// TIA Portal project "PLC_Batt" (V16)

(* hardware
DEVICE "S71500/ET200MP station_1"  S7-1500 station
   slot 0: "Rail_0"  Rack  6ES7 590-1***0-0AA0
   slot 1: "PLC_1"  CPU 1516-3 PN/DP  6ES7 516-3AN02-0AB0  V2.8
      slot 3: "CPU display_1"  6ES7591-1BA00-0AA0
      slot 32768: "PROFINET interface_1"  X1
      slot 33024: "PROFINET interface_2"  X2
      slot 33280: "DP interface_1"  X3
      slot 34817: "Virtual CP interface port_1"  Virtual CP interface port  Virtual CP interface port
DEVICE "HMI_1"  KTP700 Basic PN
   slot 0: "HMI_1"  KTP700 Basic PN  6AV2 123-2GB03-0AX0  16.0.0.0
   slot 1: "HMI_RT_1"  KTP700 Basic PN  6AV2 123-2GB03-0AX0  16.0.0.0
   slot 5: "HMI_1.IE_CP_1"  PROFINET Interface  16.0.0.0
      slot 1: "PROFINET Interface_1"  PROFINET Interface
         slot 1: "Port_1"  Port
*)

// ===== PLC "PLC_1"  CPU 1516-3 PN/DP =====

VAR_GLOBAL   // PLC tag table "inputTags"
   "batteryTesterDetector" AT %I0.0 : Bool;
   "batteryVisionDetector" AT %I0.1 : Bool;
   "Clock_Byte" AT %MB0 : Byte;
   "Clock_10Hz" AT %M0.0 : Bool;
   "Clock_5Hz" AT %M0.1 : Bool;
   "Clock_2.5Hz" AT %M0.2 : Bool;
   "Clock_2Hz" AT %M0.3 : Bool;
   "Clock_1.25Hz" AT %M0.4 : Bool;
   "Clock_1Hz" AT %M0.5 : Bool;
   "Clock_0.625Hz" AT %M0.6 : Bool;
   "Clock_0.5Hz" AT %M0.7 : Bool;
END_VAR

VAR_GLOBAL   // PLC tag table "safetyTags"
   "safetyCurtain1" AT %I1.0 : Bool;
   "safetyCurtain2" AT %I1.1 : Bool;
   "safetyCurtain3" AT %I1.2 : Bool;
   "safetyCurtain4" AT %I1.3 : Bool;
   "safetyCurtain5" AT %I1.4 : Bool;
   "safetySwitch1" AT %I2.5 : Bool;
   "safetySwitch2" AT %I2.6 : Bool;
   "safetySwitch3" AT %I2.7 : Bool;
   "warnignLamp" AT %Q1.0 : Bool;
END_VAR

DATA_BLOCK "BattTester_DB1"   // DB1
{ S7_Optimized_Access := 'TRUE' }
VERSION : 0.1
// stored: InstanceOfName BattTester
"BattTester"
BEGIN
END_DATA_BLOCK

DATA_BLOCK "VisionSystem_DB"   // DB6
{ S7_Optimized_Access := 'TRUE' }
VERSION : 0.1
// stored: InstanceOfName VisionSystem
"VisionSystem"
BEGIN
END_DATA_BLOCK

DATA_BLOCK "hmiController_DB"   // DB7
{ S7_Optimized_Access := 'TRUE' }
VERSION : 0.1
// stored: InstanceOfName hmiController
"hmiController"
BEGIN
END_DATA_BLOCK

DATA_BLOCK "daneProcesowe"   // DB8
{ S7_Optimized_Access := 'TRUE' }
VERSION : 0.1
   VAR
      visionSystem : Bool := 1;
      electricTesterSystem : Bool := 1;
      awaria : Bool;
      state : Int;
   END_VAR
BEGIN
END_DATA_BLOCK

// folder: System blocks/Program resources

DATA_BLOCK "IEC_Timer_0_DB"   // DB2
{ S7_Optimized_Access := 'TRUE' }
AUTHOR : Simatic
FAMILY : IEC
NAME : IEC_TMR
VERSION : 1.0
// stored: InstanceOfName IEC_TIMER
"IEC_TIMER"
BEGIN
END_DATA_BLOCK

DATA_BLOCK "PLC_1_Connection_DB"   // DB3
{ S7_Optimized_Access := 'TRUE' }
AUTHOR : SIMATIC
FAMILY : MC7Plus
NAME : TC_IP_v4
VERSION : 1.0
// stored: InstanceOfName TCON_IP_v4
"TCON_IP_v4"
BEGIN
   ID := 1;
   InterfaceId := 64;
   LocalPort := 2000;
END_DATA_BLOCK

DATA_BLOCK "IEC_Timer_0_DB_3"   // DB10
{ S7_Optimized_Access := 'TRUE' }
AUTHOR : Simatic
FAMILY : IEC
NAME : IEC_TMR
VERSION : 1.0
// stored: InstanceOfName IEC_TIMER
"IEC_TIMER"
BEGIN
END_DATA_BLOCK

DATA_BLOCK "IEC_Timer_0_DB_4"   // DB11
{ S7_Optimized_Access := 'TRUE' }
AUTHOR : Simatic
FAMILY : IEC
NAME : IEC_TMR
VERSION : 1.0
// stored: InstanceOfName IEC_TIMER
"IEC_TIMER"
BEGIN
END_DATA_BLOCK

DATA_BLOCK "IEC_Counter_0_DB"   // DB12
{ S7_Optimized_Access := 'TRUE' }
AUTHOR : Simatic
FAMILY : IEC
NAME : CNTR
VERSION : 1.0
// stored: InstanceOfName IEC_COUNTER
"IEC_COUNTER"
BEGIN
END_DATA_BLOCK

DATA_BLOCK "zliczaniePakietowCTU"   // DB13
{ S7_Optimized_Access := 'TRUE' }
AUTHOR : Simatic
FAMILY : IEC
NAME : CNTR
VERSION : 1.0
// stored: InstanceOfName IEC_COUNTER
"IEC_COUNTER"
BEGIN
END_DATA_BLOCK

// folder: (top level)

FUNCTION_BLOCK "BattTester"   // FB1, LAD
{ S7_Optimized_Access := 'TRUE' }
VERSION : 0.1
   VAR_INPUT
      batteryActivation : Bool;
   END_VAR
   VAR_OUTPUT
      dischargeMosfet : Bool;
      errorCode : Byte;
      finish : Bool;
      impedanceOut : Real;
      testResult : Bool;
   END_VAR
   VAR
      state : Byte := 0;
      sumOfVoltages : ULInt;
      numberOfReadingsVolts : Int;
      voltageBeforeTest : Real;
      impedance : Real;
   END_VAR
   VAR_TEMP
      batteryVoltage : Real;
      freq_to_peroid : Real;
      peroidInt : Int;
      impedanceTime : Time;
      meaonOfVoltages : ULInt;
      diffBetweenVoltages : ULInt;
      current : ULInt;
   END_VAR
   VAR CONSTANT
      timeToStart : Time := T#2s;   // czas potrzebny do uruchomienia testu po wykryciu akumulatora
      BATT_WAIT : Byte := 0;
      BATT_TEST : Byte := 1;
      BATT_AFTER_TEST : Byte := 2;
      BATT_WAIT_TO_LEAVE : Byte := 3;
      BATT_ERROR : Byte := 6;
      IMPEDANCE_TEST_FREQ : Int := 1000;
      BATT_CUT_OFF_VOLTAGE : Real := 60.0;
      BATT_MIN_VOLTAGE : Real := 40.0;
      RESISTOR_VAL : Real := 500.0;
   END_VAR
   VAR_TEMP   // added for the SCL form of the ladder/FBD networks
      _w1 : Bool;
   END_VAR
BEGIN

REGION Network 1
   // odczyt napiecia pinow baterii
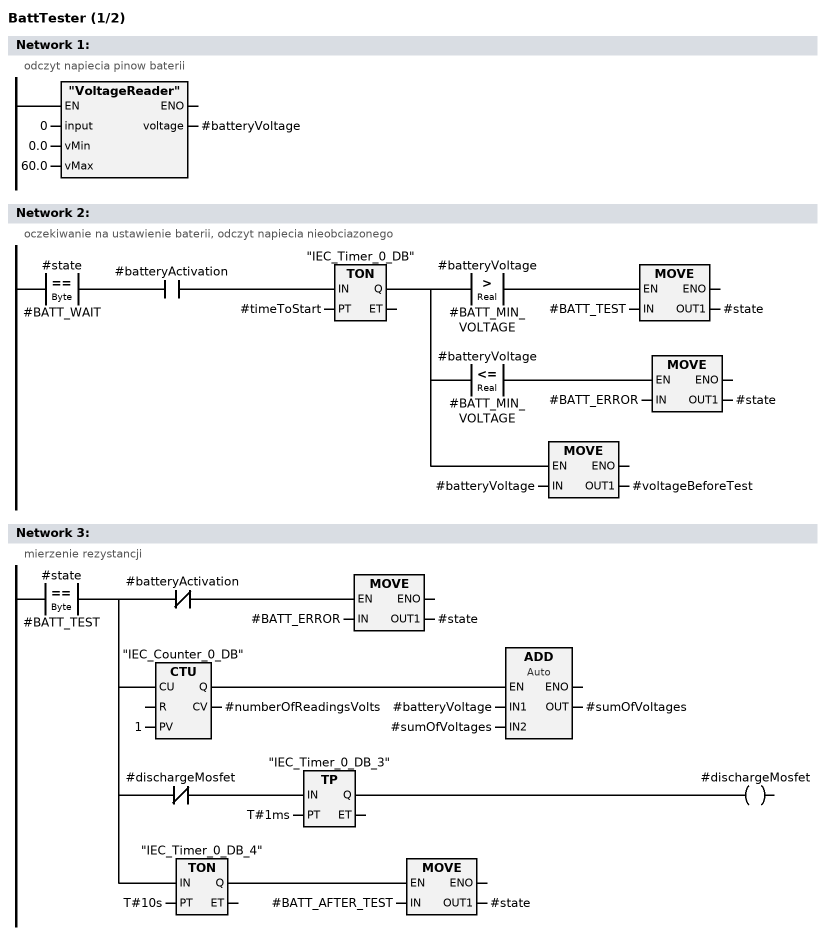
   RUNG wire#powerrail
      "VoltageReader"(input := 0, vMin := 0.0, vMax := 60.0, voltage => #batteryVoltage)
   END_RUNG
   // the same network as SCL:
   "VoltageReader"(input := 0, vMin := 0.0, vMax := 60.0, voltage => #batteryVoltage);
END_REGION

REGION Network 2
   // oczekiwanie na ustawienie baterii, odczyt napiecia nieobciazonego
   "IEC_Timer_0_DB".TON(IN := (#state = #BATT_WAIT) AND #batteryActivation, PT := #timeToStart);
   IF "IEC_Timer_0_DB".Q AND (#batteryVoltage > #BATT_MIN_VOLTAGE) THEN #state := #BATT_TEST; END_IF;
   IF "IEC_Timer_0_DB".Q AND (#batteryVoltage <= #BATT_MIN_VOLTAGE) THEN #state := #BATT_ERROR; END_IF;
   IF "IEC_Timer_0_DB".Q THEN #voltageBeforeTest := #batteryVoltage; END_IF;
END_REGION

REGION Network 3
   // mierzenie rezystancji
   #_w1 := #state = #BATT_TEST;
   IF #_w1 AND NOT #batteryActivation THEN #state := #BATT_ERROR; END_IF;
   "IEC_Counter_0_DB".CTU(CU := #_w1, PV := 1, CV => #numberOfReadingsVolts);
   IF "IEC_Counter_0_DB".Q THEN #sumOfVoltages := #batteryVoltage + #sumOfVoltages; END_IF;
   "IEC_Timer_0_DB_3".TP(IN := #_w1 AND NOT #dischargeMosfet, PT := T#1ms);
   #dischargeMosfet := "IEC_Timer_0_DB_3".Q;
   "IEC_Timer_0_DB_4".TON(IN := #_w1, PT := T#10s);
   IF "IEC_Timer_0_DB_4".Q THEN #state := #BATT_AFTER_TEST; END_IF;
END_REGION

REGION Network 4
   // wyznaczenie rezystancji wewnetrzenj ogniwa po tescie
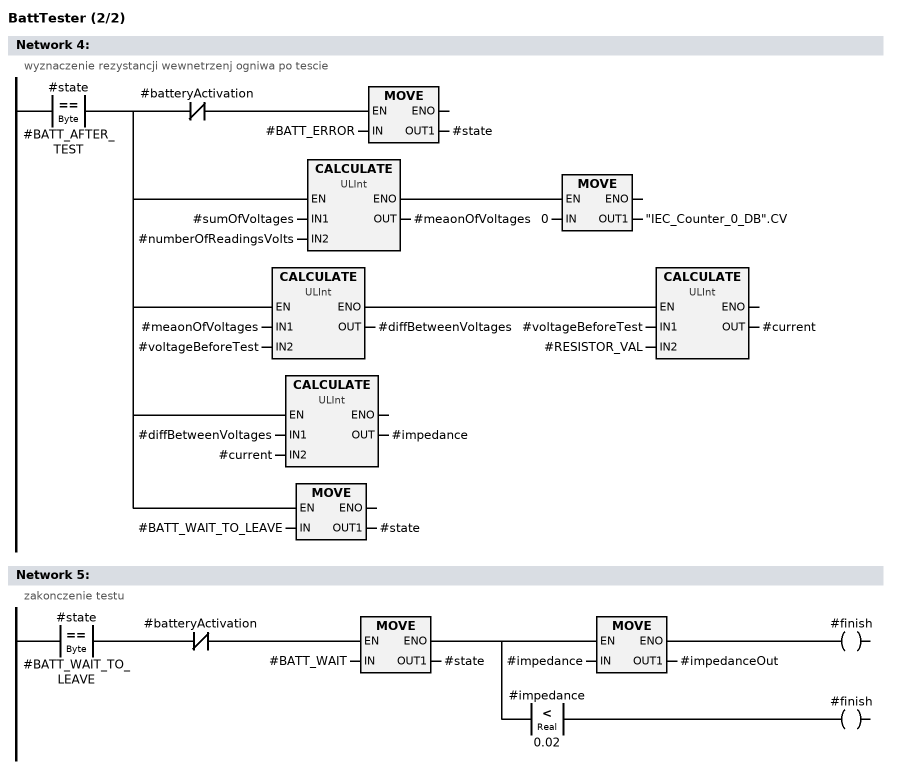
   RUNG wire#powerrail
      { S7_Templates := "SrcType := Byte" } EQ_Contact(in1 := #state, in2 := #BATT_AFTER_TEST)
      wire#w1
      I_Contact( #batteryActivation )
      Move(in := #BATT_ERROR, out1 => #state)
   END_RUNG
   RUNG wire#w1
      { S7_Templates := "SrcType := ULInt"; S7_Expression := "IN1/IN2" } Calculate(in1 := #sumOfVoltages, in2 := #numberOfReadingsVolts, out => #meaonOfVoltages)
      Move(in := 0, out1 => "IEC_Counter_0_DB".CV)
   END_RUNG
   RUNG wire#w1
      { S7_Templates := "SrcType := ULInt"; S7_Expression := "IN1 - IN2" } Calculate(in1 := #meaonOfVoltages, in2 := #voltageBeforeTest, out => #diffBetweenVoltages)
      { S7_Templates := "SrcType := ULInt"; S7_Expression := "IN1/IN2" } Calculate(in1 := #voltageBeforeTest, in2 := #RESISTOR_VAL, out => #current)
   END_RUNG
   RUNG wire#w1
      { S7_Templates := "SrcType := ULInt"; S7_Expression := "IN1 / IN2" } Calculate(in1 := #diffBetweenVoltages, in2 := #current, out => #impedance)
   END_RUNG
   RUNG wire#w1
      Move(in := #BATT_WAIT_TO_LEAVE, out1 => #state)
   END_RUNG
   // the same network as SCL:
   #_w1 := #state = #BATT_AFTER_TEST;
   IF #_w1 AND NOT #batteryActivation THEN #state := #BATT_ERROR; END_IF;
   IF #_w1 THEN
       #meaonOfVoltages := #sumOfVoltages/#numberOfReadingsVolts;
       "IEC_Counter_0_DB".CV := 0;
       #diffBetweenVoltages := #meaonOfVoltages - #voltageBeforeTest;
       #current := #voltageBeforeTest/#RESISTOR_VAL;
       #impedance := #diffBetweenVoltages / #current;
       #state := #BATT_WAIT_TO_LEAVE;
   END_IF;
END_REGION

REGION Network 5
   // zakonczenie testu
   RUNG wire#powerrail
      { S7_Templates := "SrcType := Byte" } EQ_Contact(in1 := #state, in2 := #BATT_WAIT_TO_LEAVE)
      I_Contact( #batteryActivation )
      Move(in := #BATT_WAIT, out1 => #state)
      wire#w1
      Move(in := #impedance, out1 => #impedanceOut)
      Coil( #finish )
   END_RUNG
   RUNG wire#w1
      { S7_Templates := "SrcType := Real" } LT_Contact(in1 := #impedance, in2 := 0.02)
      Coil( #finish )
   END_RUNG
   // the same network as SCL:
   #_w1 := (#state = #BATT_WAIT_TO_LEAVE) AND NOT #batteryActivation;
   IF #_w1 THEN
       #state := #BATT_WAIT;
       #impedanceOut := #impedance;
   END_IF;
   #finish := #_w1;
   #finish := #_w1 AND (#impedance < 0.02);
END_REGION
END_FUNCTION_BLOCK

FUNCTION_BLOCK "VisionSystem"   // FB2, LAD
{ S7_Optimized_Access := 'TRUE' }
VERSION : 0.1
   VAR_INPUT
      batteryDetection : Bool;
   END_VAR
   VAR_OUTPUT
      error : Bool;
      errorCode : Int;
      detectedFailedPacket : Bool;
      detectedGoodPacket : Bool;
      finished : Bool;
   END_VAR
   VAR
      TCON_Instance : TCON;
      state : Int := 1;
      batteryDetectionRisingEdge : Bool;
      recivedDataBatteryTest : Bool;
      test : Byte;
      disconnect : Bool;
      req : Bool := true;
      recv : Bool := false;
   END_VAR
   VAR_TEMP
      recivedData : Array[0..2] of Byte;
      recivedDataLen : Int;
      dataToSend : Array[0..2] of Byte;
   END_VAR
BEGIN

REGION Network 1
   // polaczenie z matlabem
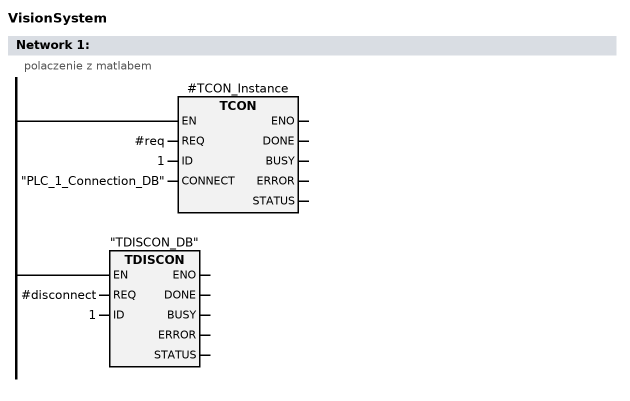
   #TCON_Instance(REQ := #req, ID := 1, CONNECT := "PLC_1_Connection_DB");   // TCON
   "TDISCON_DB"(REQ := #disconnect, ID := 1);   // TDISCON
END_REGION

REGION Network 2 (SCL)
   // maszyna stanu do testowania zgrzewów
   // maszyna stanu 
   CASE #state OF
       1: // oczekiwanie na baterie 
           IF #batteryDetection THEN
               #batteryDetectionRisingEdge := true;
               #state := 2; // zmiana stanu na 2
           END_IF;
       2: // wykryto baterie, wyslanie informacji do systemu wizyjnego 
           // wyslanie
           #dataToSend[0] := 5;
           #dataToSend[1] := 0;
           "TSEND_DB".TSEND(REQ:=TRUE,
                            ID:=1,
                            LEN:=2,
                            DATA:=#dataToSend);
           #state := 3;

       3: // odebranie i analiza odpowiedzi
           "TRCV_DB_1".TRCV(EN_R:=true,
                            ID:=1,
                            LEN:=2,
                            RCVD_LEN=>#recivedDataLen,
                            DATA:=#recivedData);
           IF #recivedDataLen > 0 THEN
               IF #recivedData[0] = 6 AND #recivedData[1] = 1 AND #finished = 0 THEN
                   #state := 4;
                   #detectedFailedPacket := 1;
                   #finished := 1;
               ELSE
                   #state := 4;
                   #detectedGoodPacket := 1;
                   #finished := 1;
               END_IF;
           END_IF;
       4: // oczekiwanie na opuszczenie baterii 
           #detectedFailedPacket := 0;
           #detectedGoodPacket := 0;
           IF #batteryDetection = false THEN
               #state := 1;
           END_IF;
   END_CASE;
END_REGION
END_FUNCTION_BLOCK

FUNCTION_BLOCK "hmiController"   // FB3, LAD
{ S7_Optimized_Access := 'TRUE' }
VERSION : 0.1
   VAR_INPUT
      batteryDetection : Bool;
      state : Int;
   END_VAR
   VAR_IN_OUT
      awaria : Bool;
   END_VAR
   VAR
      zliczaniePakietow : UDInt;
      pakietySprawne : UDInt;
      pakietyUszkodzone : UDInt;
      sprawnoscProcesu : Int;
      strState : String;
      uszkodzoneZgrzewy : UDInt;
      uszkodzoneOgniwa : UDInt;
   END_VAR
   VAR_TEMP
      awariaReset : Bool;
   END_VAR
BEGIN

REGION Network 1
   // zliczanie pakietow
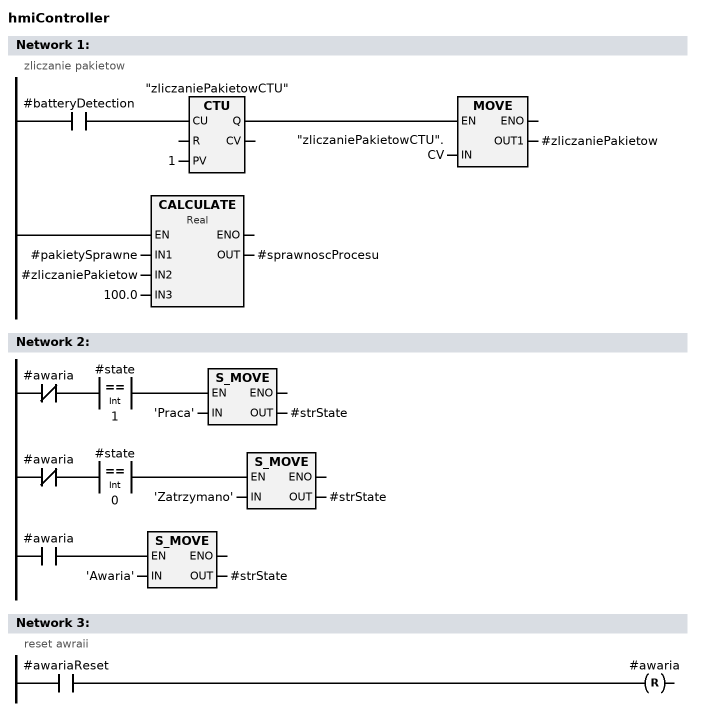
   "zliczaniePakietowCTU".CTU(CU := #batteryDetection, PV := 1);
   IF "zliczaniePakietowCTU".Q THEN #zliczaniePakietow := "zliczaniePakietowCTU".CV; END_IF;
   #sprawnoscProcesu := (#pakietySprawne / #zliczaniePakietow) * 100.0;
END_REGION

REGION Network 2
   RUNG wire#powerrail
      I_Contact( #awaria )
      { S7_Templates := "SrcType := Int" } EQ_Contact(in1 := #state, in2 := 1)
      S_Move(in := 'Praca', out => #strState)
   END_RUNG
   RUNG wire#powerrail
      I_Contact( #awaria )
      { S7_Templates := "SrcType := Int" } EQ_Contact(in1 := #state, in2 := 0)
      S_Move(in := 'Zatrzymano', out => #strState)
   END_RUNG
   RUNG wire#powerrail
      Contact( #awaria )
      S_Move(in := 'Awaria', out => #strState)
   END_RUNG
   // the same network as SCL:
   IF NOT #awaria AND (#state = 1) THEN #strState := 'Praca'; END_IF;
   IF NOT #awaria AND (#state = 0) THEN #strState := 'Zatrzymano'; END_IF;
   IF #awaria THEN #strState := 'Awaria'; END_IF;
END_REGION

REGION Network 3
   // reset awraii
   RUNG wire#powerrail
      Contact( #awariaReset )
      R_Coil( #awaria )
   END_RUNG
   // the same network as SCL:
   IF #awariaReset THEN #awaria := FALSE; END_IF;
END_REGION
END_FUNCTION_BLOCK

FUNCTION "VoltageReader" : Void   // FC1, LAD
{ S7_Optimized_Access := 'TRUE' }
VERSION : 0.1
   VAR_INPUT
      input : DInt;
      vMin : Real;
      vMax : Real;
   END_VAR
   VAR_OUTPUT
      voltage : Real;
   END_VAR
   VAR_TEMP
      tempVoltage : Real;
   END_VAR
BEGIN

REGION Network 1
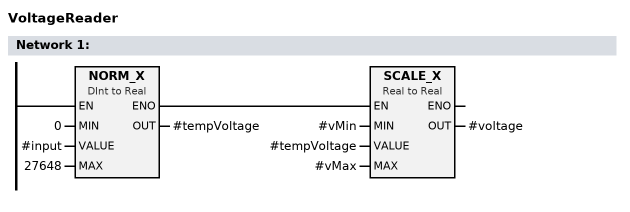
   RUNG wire#powerrail
      { S7_Templates := "[SrcType := DInt, DestType := Real]" } Normalize(min := 0, value := #input, max := 27648, out => #tempVoltage)
      { S7_Templates := "[SrcType := Real, DestType := Real]" } Scale(min := #vMin, value := #tempVoltage, max := #vMax, out => #voltage)
   END_RUNG
   // the same network as SCL:
   #tempVoltage := NORM_X(MIN := 0, VALUE := #input, MAX := 27648);
   #voltage := SCALE_X(MIN := #vMin, VALUE := #tempVoltage, MAX := #vMax);
END_REGION
END_FUNCTION

ORGANIZATION_BLOCK "Main"   // OB1, LAD, ProgramCycle
TITLE = "Main Program Sweep (Cycle)"
{ S7_Optimized_Access := 'TRUE' }
VERSION : 0.1
   VAR_INPUT
      Initial_Call : Bool;   // Initial call of this OB
      Remanence : Bool;   // =True, if remanent data are available
   END_VAR
   VAR_TEMP
      visionGoodBatt : Bool;
      visionFailBatt : Bool;
      finished : Bool;
   END_VAR
   VAR_TEMP   // added for the SCL form of the ladder/FBD networks
      _w1 : Bool;
      _w2 : Bool;
   END_VAR
BEGIN

REGION Network 1
   // system do testowania paramterów elektrycznych
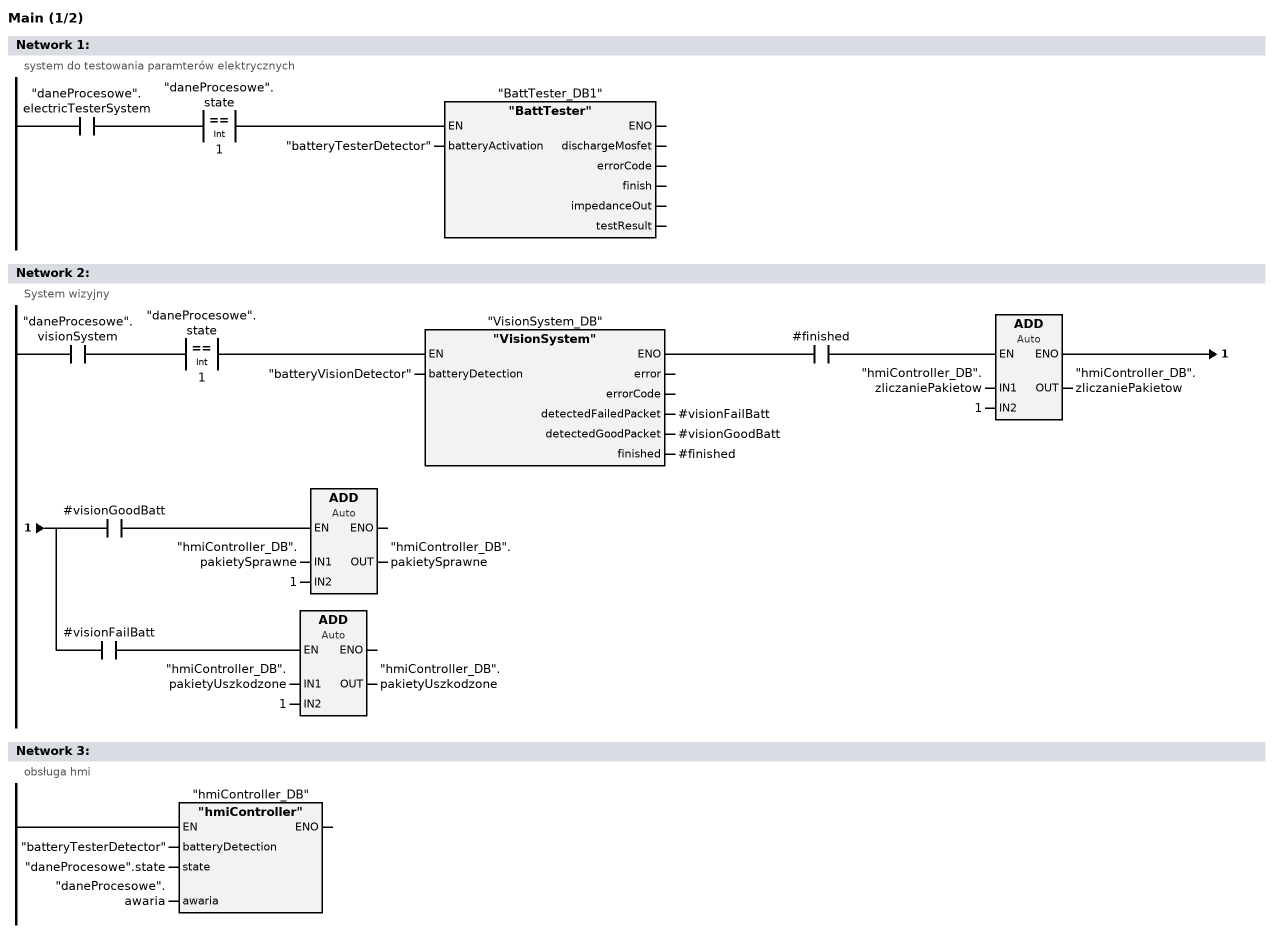
   RUNG wire#powerrail
      Contact( "daneProcesowe".electricTesterSystem )
      { S7_Templates := "SrcType := Int" } EQ_Contact(in1 := "daneProcesowe".state, in2 := 1)
      "BattTester_DB1"(batteryActivation := "batteryTesterDetector", dischargeMosfet =>, errorCode =>, finish =>, impedanceOut =>, testResult =>)
   END_RUNG
   // the same network as SCL:
   IF "daneProcesowe".electricTesterSystem AND ("daneProcesowe".state = 1) THEN
       "BattTester_DB1"(batteryActivation := "batteryTesterDetector");   // "BattTester"
   END_IF;
END_REGION

REGION Network 2
   // System wizyjny
   RUNG wire#powerrail
      Contact( "daneProcesowe".visionSystem )
      { S7_Templates := "SrcType := Int" } EQ_Contact(in1 := "daneProcesowe".state, in2 := 1)
      "VisionSystem_DB"(batteryDetection := "batteryVisionDetector", error =>, errorCode =>, detectedFailedPacket => #visionFailBatt, detectedGoodPacket => #visionGoodBatt, finished => #finished)
      Contact( #finished )
      Add(in1 := "hmiController_DB".zliczaniePakietow, in2 := 1, out => "hmiController_DB".zliczaniePakietow)
      wire#w1
      Contact( #visionGoodBatt )
      Add(in1 := "hmiController_DB".pakietySprawne, in2 := 1, out => "hmiController_DB".pakietySprawne)
   END_RUNG
   RUNG wire#w1
      Contact( #visionFailBatt )
      Add(in1 := "hmiController_DB".pakietyUszkodzone, in2 := 1, out => "hmiController_DB".pakietyUszkodzone)
   END_RUNG
   // the same network as SCL:
   "VisionSystem_DB"(EN := "daneProcesowe".visionSystem AND ("daneProcesowe".state = 1),   // "VisionSystem"
                     batteryDetection := "batteryVisionDetector",
                     detectedFailedPacket => #visionFailBatt,
                     detectedGoodPacket => #visionGoodBatt,
                     finished => #finished,
                     ENO => #_w1);
   #_w2 := #_w1 AND #finished;
   IF #_w2 THEN "hmiController_DB".zliczaniePakietow := "hmiController_DB".zliczaniePakietow + 1; END_IF;
   IF #_w2 AND #visionGoodBatt THEN
       "hmiController_DB".pakietySprawne := "hmiController_DB".pakietySprawne + 1;
   END_IF;
   IF #_w2 AND #visionFailBatt THEN
       "hmiController_DB".pakietyUszkodzone := "hmiController_DB".pakietyUszkodzone + 1;
   END_IF;
END_REGION

REGION Network 3
   // obsługa hmi
   RUNG wire#powerrail
      "hmiController_DB"(batteryDetection := "batteryTesterDetector", state := "daneProcesowe".state, awaria := "daneProcesowe".awaria)
   END_RUNG
   // the same network as SCL:
   "hmiController_DB"(batteryDetection := "batteryTesterDetector",   // "hmiController"
                      state := "daneProcesowe".state,
                      awaria := "daneProcesowe".awaria);
END_REGION

REGION Network 4
   // system bezpieczenstwa
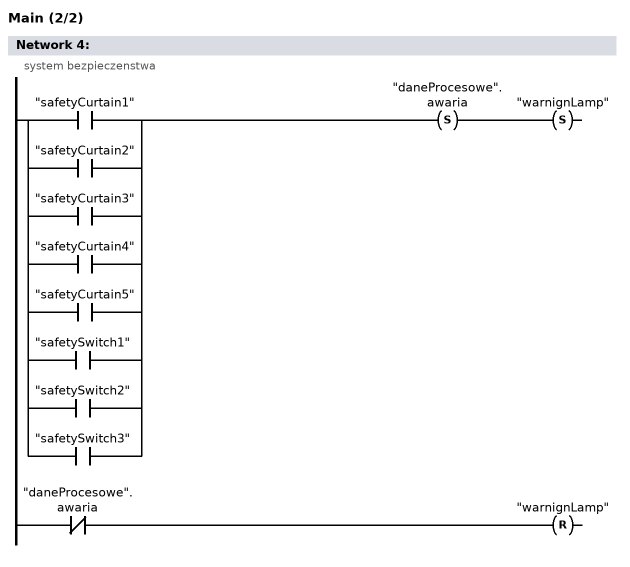
   RUNG wire#powerrail
      Contact( "safetyCurtain1" )
      wire#w1
      S_Coil( "daneProcesowe".awaria )
      S_Coil( "warnignLamp" )
   END_RUNG
   RUNG wire#powerrail
      Contact( "safetyCurtain2" )
   END_RUNG wire#w1
   RUNG wire#powerrail
      Contact( "safetyCurtain3" )
   END_RUNG wire#w1
   RUNG wire#powerrail
      Contact( "safetyCurtain4" )
   END_RUNG wire#w1
   RUNG wire#powerrail
      Contact( "safetyCurtain5" )
   END_RUNG wire#w1
   RUNG wire#powerrail
      Contact( "safetySwitch1" )
   END_RUNG wire#w1
   RUNG wire#powerrail
      Contact( "safetySwitch2" )
   END_RUNG wire#w1
   RUNG wire#powerrail
      Contact( "safetySwitch3" )
   END_RUNG wire#w1
   RUNG wire#powerrail
      I_Contact( "daneProcesowe".awaria )
      R_Coil( "warnignLamp" )
   END_RUNG
   // the same network as SCL:
   IF "safetyCurtain1" OR "safetyCurtain2" OR "safetyCurtain3" OR "safetyCurtain4" OR "safetyCurtain5" OR "safetySwitch1" OR "safetySwitch2" OR "safetySwitch3" THEN
       "daneProcesowe".awaria := TRUE;
       "warnignLamp" := TRUE;
   END_IF;
   IF NOT "daneProcesowe".awaria THEN "warnignLamp" := FALSE; END_IF;
END_REGION
END_ORGANIZATION_BLOCK

(* ===== HMI "HMI_RT_1" =====
system functions are stored by id; their names below are inferred from use
connection "HMI_Connection_1": ETHERNET, SMART_S7_1500_OMS

HMI tags "Default tag table"
   "Tag_ScreenNumber" : UInt, internal
   "daneProcesowe_visionSystem" : Bool = PLC daneProcesowe.visionSystem, 1 s
   "daneProcesowe_electricTesterSystem" : Bool = PLC daneProcesowe.electricTesterSystem, 1 s
   "daneProcesowe_state" : Int = PLC daneProcesowe.state, 1 s
   "daneProcesowe_awaria" : Bool = PLC daneProcesowe.awaria, 1 s
   "hmiController_DB_strState" : String[254] = PLC hmiController_DB.strState, 1 s
   "hmiController_DB_zliczaniePakietow" : UDInt = PLC hmiController_DB.zliczaniePakietow, 1 s
   "hmiController_DB_pakietyUszkodzone" : UDInt = PLC hmiController_DB.pakietyUszkodzone, 1 s
   "hmiController_DB_pakietySprawne" : UDInt = PLC hmiController_DB.pakietySprawne, 1 s
   "hmiController_DB_sprawnoscProcesu" : Int = PLC hmiController_DB.sprawnoscProcesu, 1 s
   "hmiController_DB_uszkodzoneZgrzewy" : UDInt = PLC hmiController_DB.uszkodzoneZgrzewy, 1 s
   "hmiController_DB_uszkodzoneOgniwa" : UDInt = PLC hmiController_DB.uszkodzoneOgniwa, 1 s

Template "Template_1" 800x480
   Button "Exit" at 714,429 size 71x50; TextOff 'Exit'; PictureOff "ExitRuntime_KTP700_Basic_PN_TR"; PictureOn "ExitRuntime_KTP700_Basic_PN_TR"
      on Release: StopRuntime(0)
   Button "Template_Button" at 611,430 size 84x50; TextOff 'Ustawienia'
      on Activate: ActivateScreen("ustawienia", 0)
   Button "Template_Button_1" at 514,429 size 71x50; TextOff 'Statystyki'
      on Activate: ActivateScreen("statystyki", 0)
   Button "Template_Button_2" at 414,429 size 71x50; TextOff 'Text'
   Button "Template_Button_3" at 314,429 size 71x50; TextOff 'Text'
   Button "Template_Button_4" at 214,429 size 71x50; TextOff 'Text'
   Button "Template_Button_5" at 114,429 size 71x50; TextOff 'Text'
   Button "Start screen" at 14,429 size 71x50; TextOff 'Start screen'; PictureOff "NavigateHome_KTP700_Basic_PN_TR"; PictureOn "NavigateHome_KTP700_Basic_PN_TR"
      on Release: ActivateScreen("Root screen", 0)
   DateTimeField "HmiScreenItemData" at 695,25 size 105x25
   DateTimeField "HmiScreenItemData_1" at 695,0 size 105x25
   TextField "Template_Text field_1" at 14,12 size 123x23; Text 'Stan maszyny:'
   IOField "Template_I/O field_1" at 142,12 size 181x32; FormatPattern ????????????????????????????????????????????????????????????????????????????????
      ProcessValue <- "hmiController_DB_strState"

screen "Root screen" 800x480, template "Template_1"
   on GenerateScreen: SetTag("Tag_ScreenNumber", 1)
   Button "Button_1" at 656,142 size 96x32; TextOff 'Zatrzymaj'
      on Click: SetTag("daneProcesowe_state", 0)
   Button "Button_2" at 657,95 size 96x32; TextOff 'Uruchom'
      on Click: SetTag("daneProcesowe_state", 1)
   Button "Button_3" at 651,186 size 111x32; TextOff 'Reset awarii'
      on Click: ResetBit("daneProcesowe_awaria")

screen "ustawienia" 800x480, template "szab1"
   Switch "Switch_1" at 638,78 size 116x34; CaptionText 'Switch'; TextOff 'OFF'; TextOn 'ON'
      ProcessValue <- "daneProcesowe_visionSystem"
   TextField "Text field_1" at 33,71 size 193x33; Text 'System wizyjny'
   Switch "Switch_2" at 640,150 size 114x34; TextOn 'ON'; CaptionText 'Switch'; TextOff 'OFF'
      ProcessValue <- "daneProcesowe_electricTesterSystem"
   TextField "Text field_2" at 32,144 size 332x33; Text 'Testy elektryczne pakietów'

Template "szab1" 800x480
   DateTimeField "HmiScreenItemData" at 695,25 size 105x25
   DateTimeField "HmiScreenItemData_1" at 695,0 size 105x25
   Button "Exit" at 714,429 size 71x50; TextOn 'Exit'; TextOff 'Exit'; PictureOn "ExitRuntime_KTP700_Basic_PN_TR"; PictureOff "ExitRuntime_KTP700_Basic_PN_TR"
      on Release: StopRuntime(0)
   Button "Start screen" at 14,429 size 71x50; TextOn 'Start screen'; TextOff 'Start screen'; PictureOn "NavigateHome_KTP700_Basic_PN_TR"; PictureOff "NavigateHome_KTP700_Basic_PN_TR"
      on Release: ActivateScreen("Root screen", 0)

screen "statystyki" 800x480, template "szab1"
   IOField "I/O field_1" at 235,55 size 96x32; FormatPattern 9999999999
      ProcessValue <- "hmiController_DB_zliczaniePakietow"
   TextField "Text field_1" at 40,55 size 156x23; Text 'Wykonane pakiety'
   IOField "I/O field_2" at 234,97 size 96x32; FormatPattern 9999999999
      ProcessValue <- "hmiController_DB_pakietyUszkodzone"
   TextField "Text field_2" at 42,98 size 169x23; Text 'Uszkodzone pakiety'
   TextField "Text field_3" at 11,22 size 62x23; Text 'Ogólne'
   IOField "I/O field_3" at 235,141 size 96x32; FormatPattern 9999999999
      ProcessValue <- "hmiController_DB_pakietySprawne"
   TextField "Text field_4" at 42,142 size 142x23; Text 'Sprawne pakiety'
   IOField "I/O field_4" at 235,184 size 92x32; FormatPattern s99999
      ProcessValue <- "hmiController_DB_sprawnoscProcesu"
   TextField "Text field_5" at 42,185 size 160x23; Text 'Sprawność procesu'
   TextField "Text field_6" at 359,76 size 169x23; Text 'Statystki uszkodzeń'
   IOField "I/O field_5" at 696,145 size 96x32; FormatPattern 9999999999
      ProcessValue <- "hmiController_DB_uszkodzoneZgrzewy"
   TextField "Text field_7" at 359,151 size 295x23; Text 'Pakiety z uszkodzonymi zgrzewami'
   IOField "I/O field_6" at 696,183 size 96x32; FormatPattern 9999999999
      ProcessValue <- "hmiController_DB_uszkodzoneOgniwa"
   TextField "Text field_8" at 363,189 size 285x23; Text 'Pakiety z uszkodzonymi ogniwami'
*)